(* CODESYS project ST_SEQUENCE_LOGIC.project

Project tree, tasks and I/O mapping:
  Device : AC702, Shenzhen Inovance Technology Co., Ltd., version 3.5.11.51
    application Application
      libraries: Standard, * (System)
      task MainTask (cyclic, interval 20 ms, priority 2) calls PLC_PRG
      program SEQ [ST]
      DifferentialMonitor
      program PLC_PRG [ST]
    HardWare Configuration
    Network Configuration
    Device Diagnosis
    Resources List
    ConfigStorage
    SoftMotion General Axis Pool
    LocalHSIO : 本地高速IO, 汇川技术股份有限公司, version 1.0.0.0
        unmapped channels: DigitalInput, DigitalOutput
    MODBUS_TCP : ModbusTCP本地从站, inovance, version 00.00.00.10
    HwConfiguratioinDevice : SystemConfig, Inovance, version 00.00.00.10
        settings: NetworkConfigArray.NetworkConfigArray.BusType = 10; NetworkConfigArray.NetworkConfigArray.RackSum = 1; NetworkConfigArray.NetworkConfigArray.HardwareConfigArray.HardwareConfigArray.RackNo = 1
*)

// Device/Application/PLC_PRG
PROGRAM PLC_PRG
VAR
	newVar: BOOL;
END_VAR

SEQ(iResetPB:=FALSE, iStartPB:=TRUE, iCylinderRetracted:=TRUE,
	iPartSensor:=TRUE, iCylinderExtended:=TRUE, iClampSensorClosed:=TRUE);

END_PROGRAM

// Device/Application/SEQ
PROGRAM SEQ
VAR_INPUT
	iResetPB: BOOL;
END_VAR
VAR
	step: INT;
	faulted: BOOL := FALSE;
	stepTimer: TON;
	oClampValve: BOOL := FALSE;
	oWorkCylinder: BOOL := FALSE;
	oCycleActiveLamp: BOOL := FALSE;
	oFaultLamp: BOOL := FALSE;
	timerEnable: BOOL := FALSE;
END_VAR
VAR_INPUT
	iStartPB: BOOL;
	iPartSensor: BOOL;
END_VAR
VAR
	timerPreset: TIME := T#5S;
END_VAR
VAR_INPUT
	iClampSensorClosed: BOOL;
	iCylinderExtended: BOOL;
	iCylinderRetracted: BOOL;
END_VAR

IF iResetPB THEN
    step := 0;
    faulted := FALSE;
END_IF;

// --- Fault Handling ---
IF faulted THEN
    step := 99; // Go to a fault step
END_IF;

// --- Step Timer Instance ---
// The timer is enabled when necessary in specific steps.
// Preset time (PT) can also be adjusted per step if needed before enabling.
stepTimer(IN:=timerEnable, PT:=timerPreset);

// --- Main Sequence CASE Statement ---
CASE step OF
    // ----- Step 0: Idle / Waiting for Start -----
    0:
        // Actions
        oClampValve := FALSE;
        oWorkCylinder := FALSE;
        oCycleActiveLamp := FALSE;
        oFaultLamp := faulted; // Show fault if reset hasn't occurred
        timerEnable := FALSE;
        faulted := FALSE; // Clear fault flag once acknowledged (or on explicit reset)

        // Transition
        IF iStartPB AND iPartSensor AND NOT faulted THEN
            step := 10;
        END_IF;

    // ----- Step 10: Clamp the Part -----
    10:
        // Actions
        oCycleActiveLamp := TRUE;
        oClampValve := TRUE;
        timerPreset := TIME#3S; // Set timeout for clamping action
        timerEnable := TRUE;

        // Transition
        IF iClampSensorClosed THEN
            step := 20;
            timerEnable := FALSE; // Disable timer, action complete
        END_IF;

        // Timeout Check
        IF stepTimer.Q THEN
            faulted := TRUE;
            timerEnable := FALSE; // Disable timer on fault
        END_IF;

    // ----- Step 20: Extend Work Cylinder -----
    20:
        // Actions
        oWorkCylinder := TRUE;
        timerPreset := TIME#5S; // Set timeout for extension
        timerEnable := TRUE;

        // Transition
        IF iCylinderExtended THEN
            step := 30;
            timerEnable := FALSE;
        END_IF;

        // Timeout Check
        IF stepTimer.Q THEN
            faulted := TRUE;
            timerEnable := FALSE;
        END_IF;

    // ----- Step 30: Retract Work Cylinder -----
    30:
        // Actions
        oWorkCylinder := FALSE;
        timerPreset := TIME#5S; // Set timeout for retraction
        timerEnable := TRUE;

        // Transition
        IF iCylinderRetracted THEN
            step := 40;
            timerEnable := FALSE;
        END_IF;

        // Timeout Check
        IF stepTimer.Q THEN
            faulted := TRUE;
            timerEnable := FALSE;
        END_IF;

    // ----- Step 40: Unclamp the Part -----
    40:
        // Actions
        oClampValve := FALSE;
        timerPreset := TIME#3S; // Set timeout for unclamping
        timerEnable := TRUE;

        // Transition
        IF NOT iClampSensorClosed THEN // Wait for clamp to open
            step := 0; // Sequence complete, return to Idle
            timerEnable := FALSE;
        END_IF;

        // Timeout Check
        IF stepTimer.Q THEN
            faulted := TRUE;
            timerEnable := FALSE;
        END_IF;

   // ----- Step 99: Fault State -----
   99:
        // Actions
        oClampValve := FALSE;
        oWorkCylinder := FALSE;
        oCycleActiveLamp := FALSE;
        oFaultLamp := TRUE;
        timerEnable := FALSE;
        // Requires iResetPB to exit this state (handled by global reset logic)

ELSE // Default case, should not be reached in normal operation
    step := 0;
    faulted := TRUE; // Indicate an unexpected state

END_CASE;

END_PROGRAM
